{attribute 'GeneratedUsingTerminal: EL5152-0000-0018'}
{attribute addProperty BoxType "EL5152-0000-0018"}
{attribute addProperty Id "EtcSlaveTerminalBaseENC_Status_compact_Channel_1AT %I*ENC_Status_compact_Channel_FA024B168ENC_Period_Channel_1AT %I*ENC_Period_Channel_24B63C534ENC_Status_compact_Channel_2AT %I*ENC_Status_compact_Channel_FA024B168ENC_Period_Channel_2AT %I*ENC_Period_Channel_24B63C534ENC_Control_compact_Channel_1AT %Q*ENC_Control_compact_Channel_2ED727EF3ENC_Control_compact_Channel_2AT %Q*ENC_Control_compact_Channel_2ED727EF3WcStateAT %I*WcState_9091E0EB2InfoDataAT %I*InfoData_32EB74EA10"}
{attribute addProperty CRC "3055333358"}
{attribute addProperty Size "42"}
TYPE EL5152_B61CAFEE EXTENDS EtcSlaveTerminalBase :
STRUCT
	{attribute addProperty Name "ENC_Status_compact_Channel_1"}
	ENC_Status_compact_Channel_1 : ENC_Status_compact_Channel_FA024B16;
	{attribute addProperty Name "ENC_Period_Channel_1"}
	ENC_Period_Channel_1 : ENC_Period_Channel_24B63C53;
	{attribute addProperty Name "ENC_Status_compact_Channel_2"}
	ENC_Status_compact_Channel_2 : ENC_Status_compact_Channel_FA024B16;
	{attribute addProperty Name "ENC_Period_Channel_2"}
	ENC_Period_Channel_2 : ENC_Period_Channel_24B63C53;
	{attribute addProperty Name "ENC_Control_compact_Channel_1"}
	ENC_Control_compact_Channel_1 : ENC_Control_compact_Channel_2ED727EF;
	{attribute addProperty Name "ENC_Control_compact_Channel_2"}
	ENC_Control_compact_Channel_2 : ENC_Control_compact_Channel_2ED727EF;
	{attribute addProperty Name "WcState"}
	WcState : WcState_9091E0EB;
	{attribute addProperty Name "InfoData"}
	InfoData : InfoData_32EB74EA;
END_STRUCT
END_TYPE

(* stored: Version 1.2.0.0, ProductVersion 3.1.4024.9
   DUT EL5152_B61CAFEE: Id {e4844f26-9770-489e-956b-7b1a83c8dba9} *)
